// Mitsubishi GX Works2 project: master   PLC: Q00

// global labels: Global1
VAR_GLOBAL
  iTank_glob AT D0 : INT;
  iPådragUt_glob AT D10 : INT;  (* generelt pådrag *)
  iPådragInn_glob AT D12 : INT;
  bModus_glob AT M23 : BOOL;  (* frekvensomformer eller ventil *)
  FO_flow_glob AT D11 : INT;  (* pådrag fra frekvensomformer *)
  iReferanse_glob AT D20 : INT;  (* settverdi *)
  iKpInn_glob AT D14 : INT;
  iKiInn_glob AT D15 : INT;
  iKdInn_glob AT D16 : INT;
  bManuell_glob AT M24 : BOOL;
  iTfInn_glob AT D17 : INT;
  bVentil1_glob AT M20 : BOOL;
  bVentil2_glob AT M21 : BOOL;
  bVentil3_glob AT M22 : BOOL;
  TIL_FRA_SLAVE_1 : TIL_FRA_SLAVE;
  bResetAlarm_glob AT M25 : BOOL;
  bAlarmCritLow_glob AT M26 : BOOL;
  bAlarmLow_glob AT M27 : BOOL;
  bAlarmHigh_glob AT M28 : BOOL;
  bAlarmCritHigh_glob AT M29 : BOOL;
  bEmergency_glob AT M30 : BOOL;
  iP_glob AT D18 : INT;
  iI_glob AT D19 : INT;
  iD_glob AT D21 : INT;
  iKpAuto_glob AT D22 : INT;
  iKiAuto_glob AT D23 : INT;
  iKdAuto_glob AT D24 : INT;
  iTfAuto_glob AT D25 : INT;
  INITIERING_1 : INITIERING;
  iKff AT D28 : INT;
  iAutoCtrl AT D26 : INT;
  iNomPådrag AT D27 : INT;
  iRateSek AT D29 : INT;
  bForover_glob AT M31 : BOOL;
  bStart_glob AT M32 : BOOL;
  bStopp_glob AT M33 : BOOL;
  iFlowLmin_glob AT D32 : INT;
  bKlar_glob AT M34 : BOOL;
  bAutoTuneFerdig_glob AT M35 : BOOL;
  iModus_glob : INT;
  iSettpunkt_Kp_P_glob AT D36 : INT;
  iSettpunkt_Kp_PD_glob AT D37 : INT;
  iSettpunkt_Kd_PD_glob AT D38 : INT;
  iSettpunkt_Kp_PI_glob AT D39 : INT;
  iSettpunkt_Ki_PI_glob AT D40 : INT;
  iSettpunkt_Kp_PID_glob AT D41 : INT;
  iSettpunkt_Ki_PID_glob AT D42 : INT;
  iSettpunkt_Kd_PID_glob AT D43 : INT;
  iSettpunkt_Tf_PD_glob AT D17 : INT;
  iSettpunkt_Tf_PID_glob AT D17 : INT;
  iTest_Kp_glob AT D44 : INT;
  iTest_Ki_glob AT D45 : INT;
  iTest_Kd_glob AT D46 : INT;
  iTest_Tf_glob AT D17 : INT;
  REGULATOR_VALG_1 : REGULATOR_VALG;
  bInit_glob : BOOL;
END_VAR

PROGRAM POU_01
(* structured ladder/FBD written out as ST: instructions are called as NAME(EN, inputs, outputs); _pN, _eN, _tN stand for wires *)
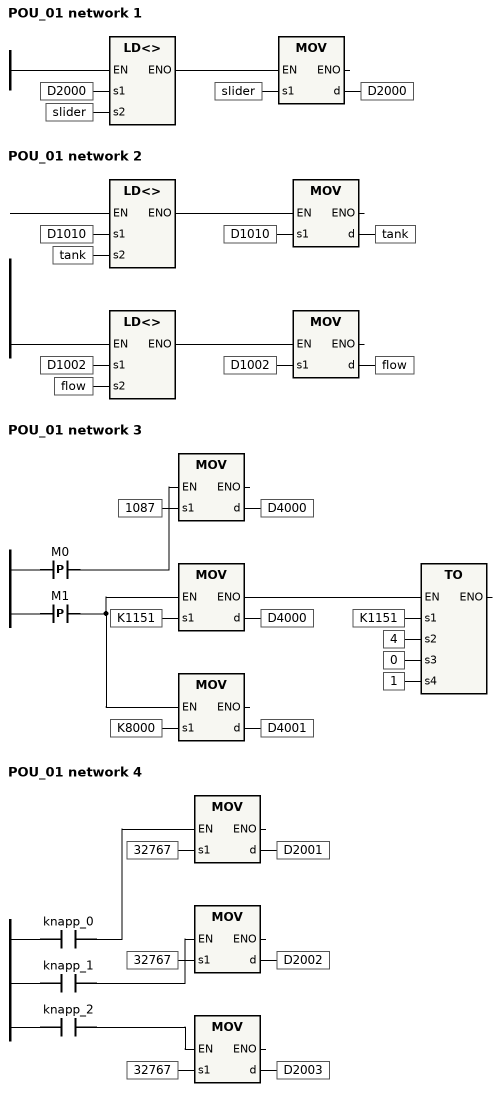
(* network 1 *)
_e1 := LD<>(TRUE, D2000, slider);
MOV(_e1, slider, D2000);
(* network 2 *)
_e1 := LD<>(TRUE, D1010, tank);
MOV(_e1, D1010, tank);
_e2 := LD<>(TRUE, D1002, flow);
MOV(_e2, D1002, flow);
(* network 3 *)
MOV(LDP(TRUE, M0), 1087, D4000);
_p1 := LDP(TRUE, M1);
_e2 := MOV(_p1, K1151, D4000);
TO(_e2, K1151, 4, 0, 1);
MOV(_p1, K8000, D4001);
(* network 4 *)
MOV(knapp_0, 32767, D2001);
MOV(knapp_1, 32767, D2002);
MOV(knapp_2, 32767, D2003);
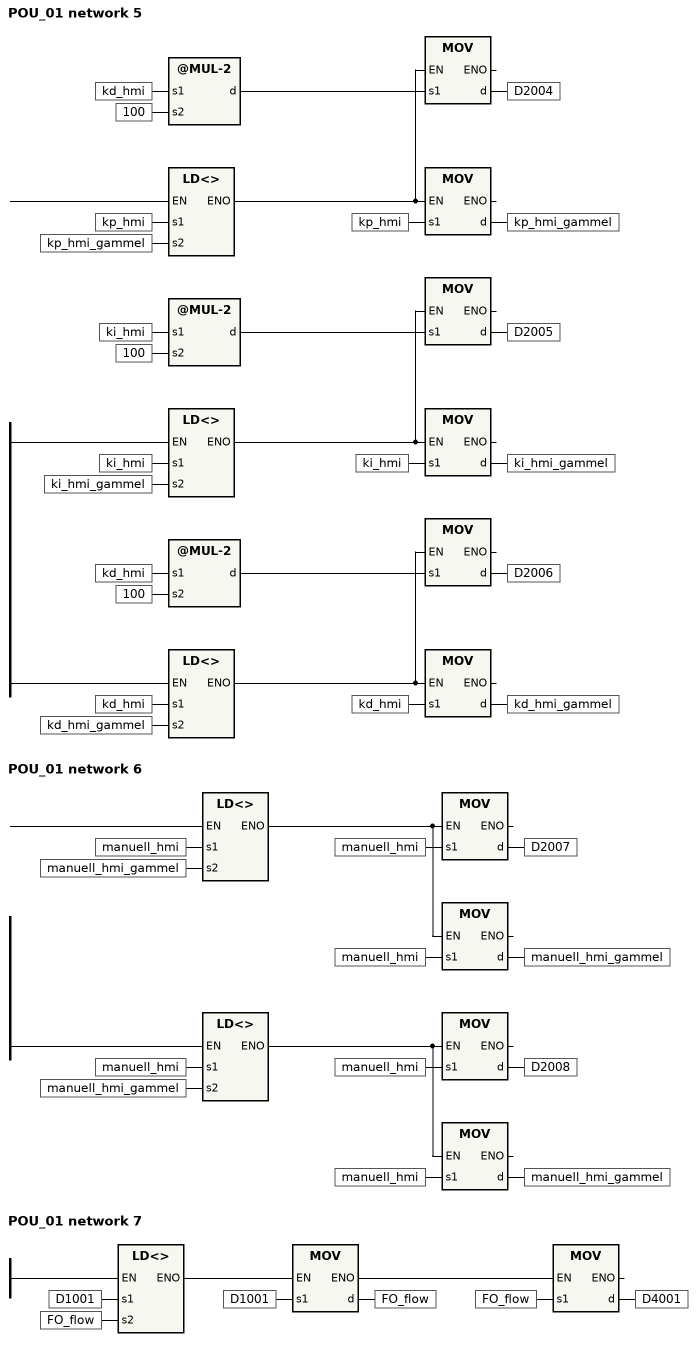
(* network 5 *)
_e1 := LD<>(TRUE, kp_hmi, kp_hmi_gammel);
MOV(_e1, @MUL-2(kd_hmi, 100), D2004);
MOV(_e1, kp_hmi, kp_hmi_gammel);
_e2 := LD<>(TRUE, ki_hmi, ki_hmi_gammel);
MOV(_e2, @MUL-2(ki_hmi, 100), D2005);
MOV(_e2, ki_hmi, ki_hmi_gammel);
_e3 := LD<>(TRUE, kd_hmi, kd_hmi_gammel);
MOV(_e3, @MUL-2(kd_hmi, 100), D2006);
MOV(_e3, kd_hmi, kd_hmi_gammel);
(* network 6 *)
_e1 := LD<>(TRUE, manuell_hmi, manuell_hmi_gammel);
MOV(_e1, manuell_hmi, D2007);
MOV(_e1, manuell_hmi, manuell_hmi_gammel);
_e2 := LD<>(TRUE, manuell_hmi, manuell_hmi_gammel);
MOV(_e2, manuell_hmi, D2008);
MOV(_e2, manuell_hmi, manuell_hmi_gammel);
(* network 7 *)
_e1 := LD<>(TRUE, D1001, FO_flow);
_e2 := MOV(_e1, D1001, FO_flow);
MOV(_e2, FO_flow, D4001);
END_PROGRAM

FUNCTION_BLOCK toggle_hmi
VAR_INPUT
  Input : BOOL;
END_VAR
VAR_OUTPUT
  FlipFlop : BOOL;
END_VAR
VAR
  OldInput : BOOL;
  oneshot : BOOL;
END_VAR
oneshot:= Input AND NOT OldInput;

IF oneshot THEN
	FlipFlop := NOT FlipFlop;
END_IF;

OldInput:=Input;
END_FUNCTION_BLOCK

FUNCTION_BLOCK TIL_FRA_SLAVE
VAR_INPUT
  iReferanse : INT;
END_VAR
VAR_OUTPUT
  iTank : INT;
  iPådragUt : INT;
END_VAR
VAR_INPUT
  bVentil1 : BOOL;
  bVentil2 : BOOL;
  bVentil3 : BOOL;
  iKp : INT;
  iKi : INT;
  iKd : INT;
  iTf : INT;
  bModus : BOOL;
  bManuell : BOOL;
END_VAR
VAR_OUTPUT
  FO_flow : INT;
END_VAR
VAR
  iKp_old : INT;
  iKi_old : INT;
  iKd_old : INT;
  iPådrag_old : INT;
  iTf_old : INT;
END_VAR
VAR_OUTPUT
  iP : INT;
  iI : INT;
  iD : INT;
  bAlarmCritLow : BOOL;
  bAlarmLow : BOOL;
  bAlarmHigh : BOOL;
  bAlarmCritHigh : BOOL;
  bEmergency : BOOL;
END_VAR
VAR_INPUT
  bResetAlarm : BOOL;
END_VAR
VAR_OUTPUT
  iKpAuto : INT;
  iKiAuto : INT;
  iKdAuto : INT;
  iTfAuto : INT;
END_VAR
VAR
  TankNy : INT;
  iAlarmWord : INT;
END_VAR
VAR_INPUT
  bForover : BOOL;
  bStart : BOOL;
  bStopp : BOOL;
END_VAR
VAR_OUTPUT
  iFlowLmin : INT;
  bKlar : BOOL;
END_VAR
VAR_INPUT
  iPådragInn : INT;
END_VAR
(* ===================== TIL SLAVE===================== *)

(* Referanse *)
MOV(TRUE, iReferanse, D2000);

(* Ventil 1 *)
D2001.0 := bVentil1;
D2001.1 := bVentil2;
D2001.2 := bVentil3;

(* Kp *)
IF iKp <> iKp_old THEN
	MOV(TRUE, iKp, D2004);
	MOV(TRUE, iKp, iKp_old);
END_IF;

(* Ki *)
IF iKi <> iKi_old THEN
	MOV(TRUE, iKi, D2005);
	MOV(TRUE, iKi, iKi_old);
END_IF;

(* Kd *)
IF iKd <> iKd_old THEN
	MOV(TRUE, iKd, D2006);
	MOV(TRUE, iKd, iKd_old);
END_IF;

(* Manuell input*)
IF iPådragInn <> iPådrag_old THEN
	MOV(TRUE, iPådragInn, D2007);
	MOV(TRUE, iPådragInn, iPådrag_old);
END_IF;

(* Tf *)
IF iTf <> iTf_old THEN
	MOV(TRUE, iTf, D2008);
	MOV(TRUE, iTf, iTf_old);
END_IF;	

(* Frekvensomformer eller ventil *)
D2001.3 := bModus;

(* Manuell eller auto modus *)
D2001.4 := bManuell;

(* Kvittering av alarm *)
D2001.5 := bResetAlarm;

(* Bruk foroverkobling *)
D2001.6 := bForover;

(* START/STOPP *)
D2001.7 := bStart;
D2001.8 := bStopp;

(* Autotuning *)
MOV(TRUE, D26, D2012);

(* Nom Pådrag *)
MOV(TRUE, D27, D2013);

(* Foroverkoblingskoeffisient *)
MOV(TRUE, D28, D2014);

(* Ratebegrensning *)
MOV(TRUE, D29, D2015);

(* ===================== FRA SLAVE===================== *)

(* Tank-nivå *)
TankNy := D1010;

IF TankNy > 0 THEN
    IF ABS(TankNy - iTank) < 20 OR iTank= 0 THEN
        iTank:= TankNy;
    END_IF;
END_IF;

(* Pådrag *)
MOV(TRUE, D1002, iPådragUt);
	
(* Frekvensomformer pådrag *)
IF D1003 <> FO_flow THEN
	MOV(TRUE, D1003, FO_flow);
	MOV(TRUE, FO_flow, D4001);
END_IF;

(* Pådrag Kp *)
IF D1004 <> iP THEN
	MOV(TRUE, D1004, iP);
END_IF;

(* Pådrag Ki *)
IF D1005 <> iI THEN
	MOV(TRUE, D1005, iI);
END_IF;

(* Pådrag Kd *)
IF D1006 <> iD THEN
	MOV(TRUE, D1006, iD);
END_IF;

(* Alarm  *)
bAlarmCritLow  := D1007.0;
bAlarmLow      := D1007.1;
bAlarmCritHigh := D1007.2;
bAlarmHigh     := D1007.3;
bEmergency     := D1007.4;
	
(* Fra autotuning *)
IF D1011 <> iKpAuto THEN
	MOV(TRUE, D1011, iKpAuto);
	bAutoTuneFerdig_glob := 1;
END_IF;
OUT_T(bAutoTuneFerdig_glob, TC2, 50);
IF TS2 THEN
    bAutoTuneFerdig_glob := 0;
END_IF;

IF D1012 <> iKiAuto THEN
	MOV(TRUE, D1012, iKiAuto);
END_IF;

IF D1013 <> iKdAuto THEN
	MOV(TRUE, D1013, iKdAuto);
END_IF;

IF D1014 <> iTfAuto THEN
	MOV(TRUE, D1014, iTfAuto);
END_IF;

(* Oppstart *)
bKlar := D1015.1;

(* Måling av utstrømning *)
IF D1001 <> iFlowLmin THEN
	MOV(TRUE, D1001, iFlowLmin);
END_IF;
END_FUNCTION_BLOCK

PROGRAM Master_Main
(* structured ladder/FBD written out as ST: instructions are called as NAME(EN, inputs, outputs); _pN, _eN, _tN stand for wires *)
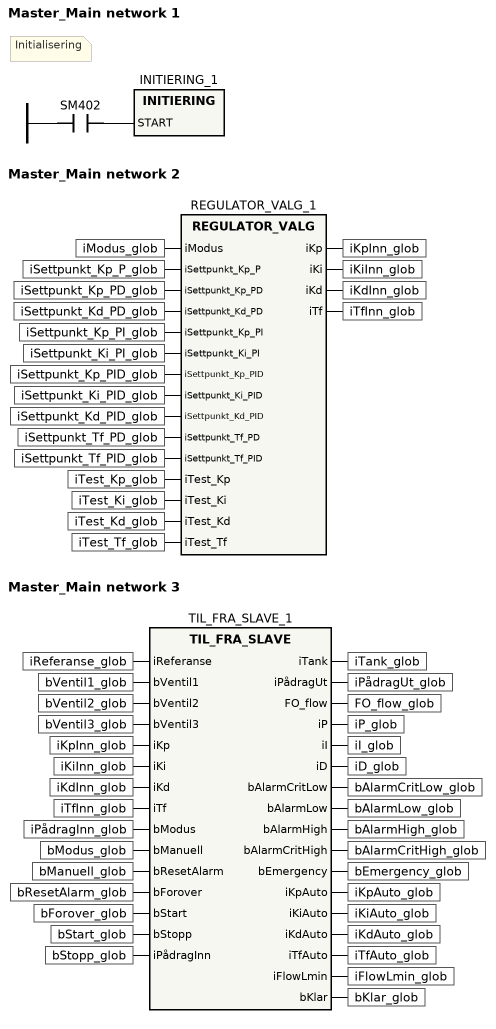
(* network 1 *)
(* Initialisering *)
INITIERING_1(START := SM402);
(* network 2 *)
REGULATOR_VALG_1(iModus := iModus_glob, iSettpunkt_Kp_P := iSettpunkt_Kp_P_glob, iSettpunkt_Kp_PD := iSettpunkt_Kp_PD_glob, iSettpunkt_Kd_PD := iSettpunkt_Kd_PD_glob, iSettpunkt_Kp_PI := iSettpunkt_Kp_PI_glob, iSettpunkt_Ki_PI := iSettpunkt_Ki_PI_glob, iSettpunkt_Kp_PID := iSettpunkt_Kp_PID_glob, iSettpunkt_Ki_PID := iSettpunkt_Ki_PID_glob, iSettpunkt_Kd_PID := iSettpunkt_Kd_PID_glob, iSettpunkt_Tf_PD := iSettpunkt_Tf_PD_glob, iSettpunkt_Tf_PID := iSettpunkt_Tf_PID_glob, iTest_Kp := iTest_Kp_glob, iTest_Ki := iTest_Ki_glob, iTest_Kd := iTest_Kd_glob, iTest_Tf := iTest_Tf_glob, iKp => iKpInn_glob, iKi => iKiInn_glob, iKd => iKdInn_glob, iTf => iTfInn_glob);
(* network 3 *)
TIL_FRA_SLAVE_1(iReferanse := iReferanse_glob, bVentil1 := bVentil1_glob, bVentil2 := bVentil2_glob, bVentil3 := bVentil3_glob, iKp := iKpInn_glob, iKi := iKiInn_glob, iKd := iKdInn_glob, iTf := iTfInn_glob, bModus := iPådragInn_glob, bManuell := bModus_glob, bResetAlarm := bManuell_glob, bForover := bResetAlarm_glob, bStart := bForover_glob, bStopp := bStart_glob, iPådragInn := bStopp_glob, iTank => iTank_glob, iPådragUt => iPådragUt_glob, FO_flow => FO_flow_glob, iP => iP_glob, iI => iI_glob, iD => iD_glob, bAlarmCritLow => bAlarmCritLow_glob, bAlarmLow => bAlarmLow_glob, bAlarmHigh => bAlarmHigh_glob, bAlarmCritHigh => bAlarmCritHigh_glob, bEmergency => bEmergency_glob, iKpAuto => iKpAuto_glob, iKiAuto => iKiAuto_glob, iKdAuto => iKdAuto_glob, iTfAuto => iTfAuto_glob, iFlowLmin => iFlowLmin_glob, bKlar => bKlar_glob);
END_PROGRAM

FUNCTION_BLOCK INITIERING
VAR_INPUT
  START : BOOL;
END_VAR
SET(START, Y00);
OUT_T(Y00, TC0, 50);
MOV(TS0, 1087, D4000);

(* Kjøres kun i første syklus etter oppstart *)
IF START THEN
    (* PID-parametere - known good verdier *)
    iKpInn_glob := 2470;
    iKiInn_glob := 78;
    iKdInn_glob := 5574;
    iTfInn_glob := 451;
    
    (* Ratebegrensning *)
    iRateSek := 5;
    
    (* Regulatormodus - start i manuell *)
    iModus_glob := 0;
    
    (* Settpunkter for hver regulatormodus *)
    iSettpunkt_Kp_P_glob := 2000;
    
    iSettpunkt_Kp_PD_glob := 2200;
    iSettpunkt_Kd_PD_glob := 4500;
    iSettpunkt_Tf_PD_glob := 400;
    
    iSettpunkt_Kp_PI_glob := 1800;
    iSettpunkt_Ki_PI_glob := 60;
    
    iSettpunkt_Kp_PID_glob := 2470;
    iSettpunkt_Ki_PID_glob := 78;
    iSettpunkt_Kd_PID_glob := 5574;
    iSettpunkt_Tf_PID_glob := 451;
    
    (* Test-verdier (for justerbar modus) - start med samme som PID *)
    iTest_Kp_glob := 2470;
    iTest_Ki_glob := 78;
    iTest_Kd_glob := 5574;
    iTest_Tf_glob := 451;
    
    (* Referanse *)
    iReferanse_glob := 50;
    
    (* Ventiler - 2 av 3 åpne ved oppstart (som oppgaven krever) *)
    bVentil1_glob := TRUE;
    bVentil2_glob := TRUE;
    bVentil3_glob := FALSE;
    
    (* Modus: ventilregulering som default *)
    bModus_glob := FALSE;
    
    (* Ikke foroverkobling som default *)
    bForover_glob := FALSE;
END_IF;
END_FUNCTION_BLOCK

FUNCTION_BLOCK REGULATOR_VALG
VAR_INPUT
  iModus : INT;
  iSettpunkt_Kp_P : INT;
  iSettpunkt_Kp_PD : INT;
  iSettpunkt_Kd_PD : INT;
  iSettpunkt_Kp_PI : INT;
  iSettpunkt_Ki_PI : INT;
  iSettpunkt_Kp_PID : INT;
  iSettpunkt_Ki_PID : INT;
  iSettpunkt_Kd_PID : INT;
  iSettpunkt_Tf_PD : INT;
  iSettpunkt_Tf_PID : INT;
  iTest_Kp : INT;
  iTest_Ki : INT;
  iTest_Kd : INT;
  iTest_Tf : INT;
END_VAR
VAR_OUTPUT
  iKp : INT;
  iKi : INT;
  iKd : INT;
  iTf : INT;
END_VAR


CASE iModus OF
    0:
        bManuell_glob := TRUE;
        
    2: (* Justerbar *)
    	bManuell_glob := FALSE;
    	iKp := iTest_Kp;
    	iKi := iTest_Ki;
    	iKd := iTest_Kd;
    	iTf := iTest_Tf;
    
    3: (* P-regulator *)
        bManuell_glob := FALSE;
        iKp := iSettpunkt_Kp_P;
        iKi := 0;
        iKd := 0;
        iTf := 0;
    
    4: (* PD-regulator *)
        bManuell_glob := FALSE;
        iKp := iSettpunkt_Kp_PD;
        iKi := 0;
        iKd := iSettpunkt_Kd_PD;
        iTf := iSettpunkt_Tf_PD;
    
    5: (* PI-regulator *)
        bManuell_glob := FALSE;
        iKp := iSettpunkt_Kp_PI;
        iKi := iSettpunkt_Ki_PI;
        iKd := 0;
        iTf := 0;
    
    6: (* PID-regulator *)
        bManuell_glob := FALSE;
        iKp := iSettpunkt_Kp_PID;
        iKi := iSettpunkt_Ki_PID;
        iKd := iSettpunkt_Kd_PID;
        iTf := iSettpunkt_Tf_PID;
END_CASE;
END_FUNCTION_BLOCK
